// TIA Portal project "Analog vattentank" (V17)

(* hardware
DEVICE "S7-1500/ET200MP station_1"  S7-1500 station
   slot 0: "Rail_0"  Rack  6ES7 590-1***0-0AA0
   slot 1: "PLC_1"  CPU 1511-1 PN  6ES7 511-1AK02-0AB0  V2.9
      slot 3: "CPU display_1"  6ES7591-1AA00-0AA0
      slot 32768: "PROFINET interface_1"  X1
         slot 32769: "Port_1"  X1 P1
         slot 32770: "Port_2"  X1 P2
      slot 34817: "Virtual CP interface port_1"  Virtual CP interface port  Virtual CP interface port
   slot 2: "DI 16x24VDC BA_1"  DI 16x24VDC BA  6ES7 521-1BH10-0AA0  V1.1
   slot 3: "DQ 16x24VDC/0.5A BA_1"  DQ 16x24VDC/0.5A BA  6ES7 522-1BH10-0AA0  V1.1
   slot 4: "AI 4xU/I/RTD/TC ST_1"  AI 4xU/I/RTD/TC ST  6ES7 531-7QD00-0AB0  V1.0
   slot 5: "AQ 4xU/I ST_1"  AQ 4xU/I ST  6ES7 532-5HD00-0AB0  V2.2
*)

// ===== PLC "PLC_1"  CPU 1511-1 PN =====

VAR_GLOBAL   // PLC tag table "IO"
   "Start" AT %I0.0 : Bool;
   "Reset" AT %I0.1 : Bool;
   "Stop" AT %I0.2 : Bool;
   "FACTORY I/O (Running)" AT %I0.3 : Bool;
   "Start light" AT %Q0.0 : Bool;
   "Reset light" AT %Q0.1 : Bool;
   "Stop light" AT %Q0.2 : Bool;
   "Level meter" AT %IW30 : Int;
   "Flow meter" AT %IW32 : Int;
   "Setpoint" AT %IW34 : Int;
   "Fill valve" AT %QW30 : Int;
   "Discharge valve" AT %QW32 : Int;
   "SP" AT %QW34 : Int;
   "PV" AT %QW36 : Int;
   "socker" AT %I2.0 : Bool;
   "vatten" AT %I2.1 : Bool;
   "honing" AT %I2.2 : Bool;
END_VAR

DATA_BLOCK "HMI start_DB"   // DB1
{ S7_Optimized_Access := 'TRUE' }
VERSION : 0.1
// stored: InstanceOfName HMI start
"HMI start"
BEGIN
END_DATA_BLOCK

DATA_BLOCK "Scalering DB"   // DB2
{ S7_Optimized_Access := 'TRUE' }
VERSION : 0.1
   VAR
      "Norm x LM" : Struct
         min : Int;   // hur hög vatten nivån är i råvärde
         max : Int := 27648;   // hur hög vatten nivån är i råvärde
         är : Int;
         bör : Int;
         "scalerat värde" : Real;
      END_STRUCT;
      "scala x LM" : Struct
         min : Int;   // skalerat värde på tankens vatten nivå
         max : Int := 300;   // skalerat värde på tankens vatten nivå
         är : Int;   // faktiska nivå på tank
         bör : Int;
      END_STRUCT;
      "morm x FV" : Struct
         min : Int;
         max : Int := 10;
         är : Int;
         bör : Int;
         "scalerat värde" : Real;
      END_STRUCT;
      "scale x FV" : Struct
         min : Int;
         max : Int := 27648;
         är : Int;
         bör : Int;
      END_STRUCT;
   END_VAR
BEGIN
END_DATA_BLOCK

DATA_BLOCK "HMI start_DB_1"   // DB4
{ S7_Optimized_Access := 'TRUE' }
VERSION : 0.1
// stored: InstanceOfName HMI start
"HMI start"
BEGIN
END_DATA_BLOCK

FUNCTION_BLOCK "HMI start"   // FB1, SCL
{ S7_Optimized_Access := 'TRUE' }
VERSION : 0.1
   VAR_INPUT
      start : Bool;
      stop : Bool;
      reset : Bool;
   END_VAR
   VAR_IN_OUT
      "stop light" : Bool;
      "start light" : Bool;
      "reset light" : Bool;
   END_VAR
BEGIN
   (*
   IF #start THEN
       #"start light" := TRUE;
       #"reset light" := FALSE;
       #"stop light" := FALSE;

   ELSIF NOT #stop THEN
       #"start light" := FALSE;
       #"reset light" := FALSE;
       #"stop light" := TRUE;

   ELSIF #reset THEN
       #"start light" := FALSE;
       #"reset light" := TRUE;
       #"stop light" := FALSE;
       // Statement section IF
       ;
   END_IF;
   *)

   IF #start THEN
       #"start light" := TRUE;
       #"stop light" := FALSE;
       #"reset light" := FALSE;
   ELSIF NOT #stop THEN
       #"start light" := FALSE;
       #"stop light" := TRUE;
       #"reset light" := FALSE;
   ELSIF #reset THEN
       #"start light" := FALSE;
       #"stop light" := FALSE;
       #"reset light" := TRUE;
       // Statement section IF
       ;
   END_IF;
END_FUNCTION_BLOCK

FUNCTION "hmi Test" : Void   // FC1, SCL
{ S7_Optimized_Access := 'TRUE' }
VERSION : 0.1
   VAR_INPUT
      start : Bool;
      stop : Bool;
      reset : Bool;
   END_VAR
   VAR_IN_OUT
      "stop light" : Bool;
   END_VAR
BEGIN
   "Start light" := TRUE;
   #"stop light" := TRUE;
END_FUNCTION

FUNCTION "scalering" : Void   // FC2, LAD
{ S7_Optimized_Access := 'TRUE' }
VERSION : 0.1
BEGIN

REGION Network 1
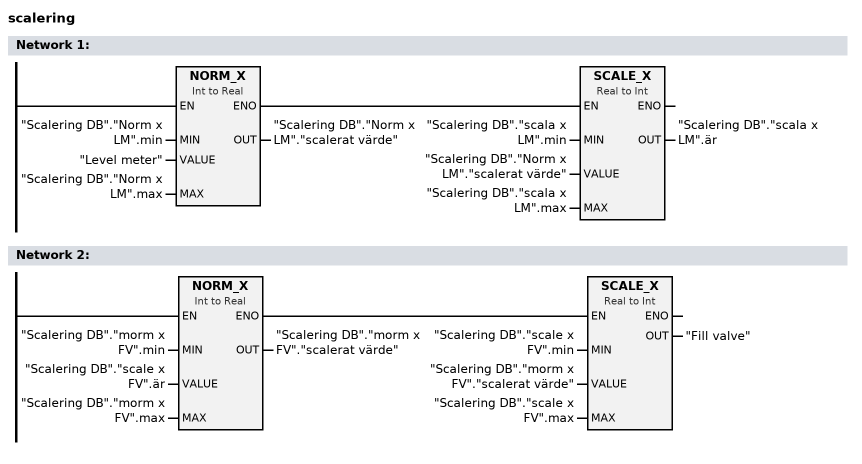
   RUNG wire#powerrail
      { S7_Templates := "[SrcType := Int, DestType := Real]" } Normalize(min := "Scalering DB"."Norm x LM".min, value := "Level meter", max := "Scalering DB"."Norm x LM".max, out => "Scalering DB"."Norm x LM"."scalerat värde")
      { S7_Templates := "[SrcType := Real, DestType := Int]" } Scale(min := "Scalering DB"."scala x LM".min, value := "Scalering DB"."Norm x LM"."scalerat värde", max := "Scalering DB"."scala x LM".max, out => "Scalering DB"."scala x LM".är)
   END_RUNG
   // the same network as SCL:
   "Scalering DB"."Norm x LM"."scalerat värde" := NORM_X(MIN := "Scalering DB"."Norm x LM".min, VALUE := "Level meter", MAX := "Scalering DB"."Norm x LM".max);
   "Scalering DB"."scala x LM".är := SCALE_X(MIN := "Scalering DB"."scala x LM".min, VALUE := "Scalering DB"."Norm x LM"."scalerat värde", MAX := "Scalering DB"."scala x LM".max);
END_REGION

REGION Network 2
   RUNG wire#powerrail
      { S7_Templates := "[SrcType := Int, DestType := Real]" } Normalize(min := "Scalering DB"."morm x FV".min, value := "Scalering DB"."scale x FV".är, max := "Scalering DB"."morm x FV".max, out => "Scalering DB"."morm x FV"."scalerat värde")
      { S7_Templates := "[SrcType := Real, DestType := Int]" } Scale(min := "Scalering DB"."scale x FV".min, value := "Scalering DB"."morm x FV"."scalerat värde", max := "Scalering DB"."scale x FV".max, out => "Fill valve")
   END_RUNG
   // the same network as SCL:
   "Scalering DB"."morm x FV"."scalerat värde" := NORM_X(MIN := "Scalering DB"."morm x FV".min, VALUE := "Scalering DB"."scale x FV".är, MAX := "Scalering DB"."morm x FV".max);
   "Fill valve" := SCALE_X(MIN := "Scalering DB"."scale x FV".min, VALUE := "Scalering DB"."morm x FV"."scalerat värde", MAX := "Scalering DB"."scale x FV".max);
END_REGION
END_FUNCTION

FUNCTION "tömma fylla" : Void   // FC3, LAD
{ S7_Optimized_Access := 'TRUE' }
VERSION : 0.1
BEGIN

REGION Network 1
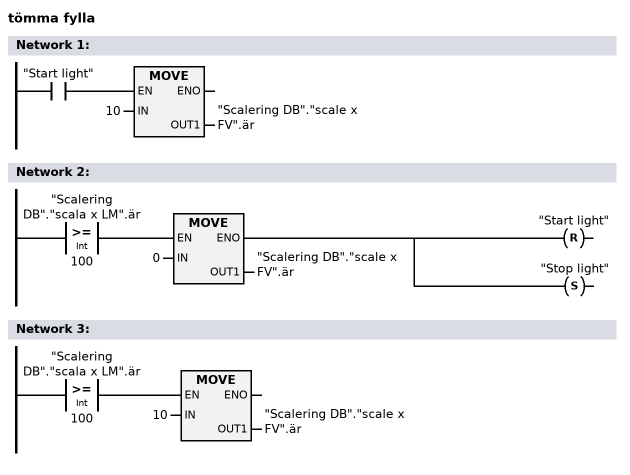
   RUNG wire#powerrail
      Contact( "Start light" )
      Move(in := 10, out1 => "Scalering DB"."scale x FV".är)
   END_RUNG
   // the same network as SCL:
   IF "Start light" THEN "Scalering DB"."scale x FV".är := 10; END_IF;
END_REGION

REGION Network 2
   RUNG wire#powerrail
      { S7_Templates := "SrcType := Int" } GE_Contact(in1 := "Scalering DB"."scala x LM".är, in2 := 100)
      Move(in := 0, out1 => "Scalering DB"."scale x FV".är)
      wire#w1
      R_Coil( "Start light" )
   END_RUNG
   RUNG wire#w1
      S_Coil( "Stop light" )
   END_RUNG
   // the same network as SCL:
   IF "Scalering DB"."scala x LM".är >= 100 THEN
       "Scalering DB"."scale x FV".är := 0;
       "Start light" := FALSE;
       "Stop light" := TRUE;
   END_IF;
END_REGION

REGION Network 3
   RUNG wire#powerrail
      { S7_Templates := "SrcType := Int" } GE_Contact(in1 := "Scalering DB"."scala x LM".är, in2 := 100)
      Move(in := 10, out1 => "Scalering DB"."scale x FV".är)
   END_RUNG
   // the same network as SCL:
   IF "Scalering DB"."scala x LM".är >= 100 THEN "Scalering DB"."scale x FV".är := 10; END_IF;
END_REGION
END_FUNCTION

ORGANIZATION_BLOCK "Main"   // OB1, LAD, ProgramCycle
TITLE = "Main Program Sweep (Cycle)"
{ S7_Optimized_Access := 'TRUE' }
VERSION : 0.1
   VAR_INPUT
      Initial_Call : Bool;   // Initial call of this OB
      Remanence : Bool;   // =True, if remanent data are available
   END_VAR
BEGIN

REGION Network 1
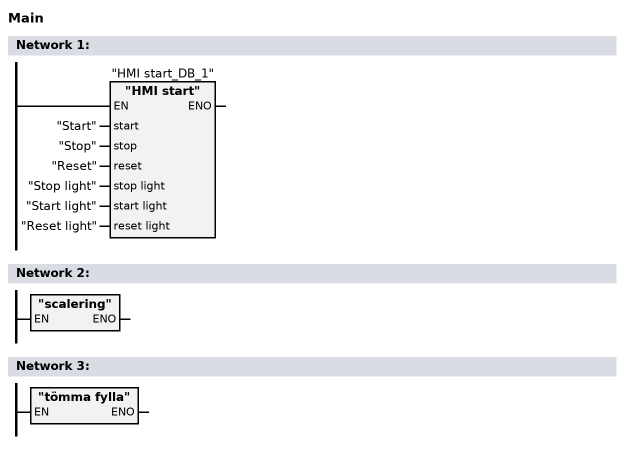
   RUNG wire#powerrail
      "HMI start_DB_1"(start := "Start", stop := "Stop", reset := "Reset", "stop light" := "Stop light", "start light" := "Start light", "reset light" := "Reset light")
   END_RUNG
   // the same network as SCL:
   "HMI start_DB_1"(start := "Start",   // "HMI start"
                    stop := "Stop",
                    reset := "Reset",
                    "stop light" := "Stop light",
                    "start light" := "Start light",
                    "reset light" := "Reset light");
END_REGION

REGION Network 2
   RUNG wire#powerrail
      "scalering"()
   END_RUNG
   // the same network as SCL:
   "scalering"();
END_REGION

REGION Network 3
   RUNG wire#powerrail
      "tömma fylla"()
   END_RUNG
   // the same network as SCL:
   "tömma fylla"();
END_REGION
END_ORGANIZATION_BLOCK